INTERFACE I_ReadableData

PROPERTY PUBLIC Data : T_MAXSTRING
GET
END_GET
END_PROPERTY

METHOD PUBLIC TryGet : BOOL;
VAR_INPUT
	Value : ANY;
END_VAR
END_METHOD

METHOD PUBLIC TryGetTo : BOOL;
VAR_INPUT
	Destination : PVOID;
	DestinationSize : UDINT;
END_VAR
END_METHOD

END_INTERFACE

(* stored: Version 1.1.0.1, ProductVersion 3.1.4024.12
   Itf I_ReadableData: Id {82e99dec-d205-085b-0b23-3522cd3d2d7e}
   Property Data: Id {b846db2d-ce55-40fe-8775-fa0fddf20325}
   Get Get: Id {60c63cf6-7384-4b53-ab8e-fcb933a9e5c7}
   Method TryGet: Id {33239db5-298f-0f43-1757-b2fb9ec949c8}
   Method TryGetTo: Id {d98c94e4-9b11-052f-047f-329220f0064f} *)
